// TwinCAT 3 PLC project Untitled1
// ProgramVersion: 3.1.4024.0
// libraries:
//   Tc2_Standard, * (Beckhoff Automation GmbH)
//   Tc2_System, * (Beckhoff Automation GmbH)
//   Tc3_Module, * (Beckhoff Automation GmbH)
// project tree:
//   / GlobalTextList.TcGTLO, PlcTask.TcTTO, Visualization Manager.TcVMO (not stored), Visualization.TcVIS
//   GVLs/ GVL.TcGVL
//   POUs/ Brightspace.TcPOU, MotivationAnalysis.TcPOU, Student.TcPOU, Calender.TcPOU
// real-time tasks:
//   TASK PlcTask: cycle T#10ms, priority 20, ADS port 350
//   TASK brightspace: cycle T#10ms, priority 1, ADS port 351
//   TASK Calender: cycle T#10ms, priority 2, ADS port 352

CONFIGURATION Untitled1
    RESOURCE PLC ON TwinCAT3
        TASK PlcTask(INTERVAL := T#10ms, PRIORITY := 20);
        PROGRAM Student WITH PlcTask : Student;
        PROGRAM Brightspace WITH PlcTask : Brightspace;
        PROGRAM Calender WITH PlcTask : Calender;
    END_RESOURCE
END_CONFIGURATION

// ---- GVLs/GVL.TcGVL
{attribute 'qualified_only'}
VAR_GLOBAL
	
	StartPls : BOOL;		//signal student to start doing something
	Day : INT:= 0;			//keeps track of what day it is
	Finished: BOOL := 0;	//student can signal he has finished an assingment
	MainDueIn: INT := 0;	//shows how far you are from the deadline
	Cycle: BOOL;			//shows daycycle
END_VAR

// ---- POUs/Student.TcPOU
PROGRAM Student		//program pretending to be a student
VAR
	MaxMotivation1: INT := 75; 	//maximum amount of motivation the student can have on a given day
	Phone: SR;					//phone saves the signal from brightspace as a notification
	StudentNotification: BOOL;	
	DontWantTo: BOOL;			//shows the student is not going to do the work
	MotTrig: R_TRIG;			
	MotTrigHigh: BOOL;
	Motivation: INT;
	Timer: TON;
	
	MotivationTracker: ARRAY[1..25] OF INT;	//tracks motivation for visualisation
	ArrayCount: INT := 1;					//position in bar graph
END_VAR

//set notification
Phone(SET1:=GVL.StartPls , RESET:=GVL.Finished OR DontWantTo , Q1=>StudentNotification );

//daily motivation calculated each morning :)
MotTrig(CLK:=StudentNotification , Q=>MotTrigHigh );
IF MotTrigHigh = TRUE THEN
	Motivation := MotivationAnalysis(MaxMotivation2:=MaxMotivation1 );
	
	//visualisation fun
	MotivationTracker[ArrayCount] := Motivation;
	ArrayCount := ArrayCount + 1;
	IF ArrayCount > 25 THEN
		ArrayCount := 1;
	END_IF
END_IF

//when the student has a notification pending they will decide what to do with it depending on the amount of motivation they have minus the amount of time they have left to finish it
IF StudentNotification = TRUE THEN
	IF (GVL.MainDueIn*-1) + Motivation > 69 THEN
		GVL.Finished := TRUE;
	ELSIF (GVL.MainDueIn*-1) + Motivation < 69 THEN
		DontWantTo := TRUE;
		Timer(IN := TRUE, PT := T#50MS);
	END_IF
END_IF

//turn DontWantTo off for as long as needed
IF Timer.Q THEN
    DontWantTo := FALSE;
    Timer(IN := FALSE);
END_IF

END_PROGRAM

// ---- POUs/MotivationAnalysis.TcPOU
FUNCTION MotivationAnalysis : INT	//function which gives a random number between 0 and the max value
VAR_INPUT
	MaxMotivation2: INT;
END_VAR
VAR
	Roll4Motivation: DRAND;
	RandomReal: LREAL;
END_VAR

//DRAND function with daynumber as seed
Roll4Motivation(Seed:=GVL.Day , Num=>RandomReal );

//changes the range from 0-1 to 1-whatever you put as maximum
MotivationAnalysis := 1 + LREAL_TO_INT (RandomReal * MaxMotivation2);

END_FUNCTION

// ---- POUs/Brightspace.TcPOU
PROGRAM Brightspace		//program pretending to be brightspace
VAR
	TaskMaster: ARRAY[1..3] OF INT := [
        0, 0, 1    // 30 day task
    ];
	TasksGiven: INT;	
	Late: BOOL;
END_VAR

//how many days till certain assignment needs to be done
GVL.MainDueIn := TaskMaster[2] - GVL.Day;

//make task
IF TaskMaster[1] = 0 OR GVL.MainDueIn < 1 AND TaskMaster[3] = 1 THEN
	GVL.Finished := FALSE;
	TaskMaster[1] := TasksGiven + 1;
	TaskMaster[2] := GVL.Day + 30;
	TaskMaster[3] := 0;
	TasksGiven := TasksGiven +1;
	GVL.StartPls := TRUE;
END_IF

//arrays and global variables dont mix
IF GVL.Finished = TRUE THEN				//yes im using this if statement as an SR flipflop
	TaskMaster[3] := 1;
END_IF
 
//send signal once to remind the student to pls start doing something
IF GVL.MainDueIn = 30 AND TaskMaster[3] = 0 OR GVL.MainDueIn = 20 AND TaskMaster[3] = 0 OR GVL.MainDueIn = 10 AND TaskMaster[3] = 0 OR GVL.MainDueIn <= 1 AND TaskMaster[3] = 0 THEN 
	GVL.StartPls := TRUE;
	IF GVL.MainDueIn <0 AND TaskMaster[3] = 0 THEN
		GVL.StartPls := GVL.Cycle;
	END_IF
ELSE
	GVL.StartPls := FALSE;		
END_IF 

IF GVL.MainDueIn <0 THEN
	Late := TRUE;
ELSE 
	Late := FALSE;
END_IF

END_PROGRAM

// ---- POUs/Calender.TcPOU
PROGRAM Calender //adjustable on/off timer program
VAR
	DayNight: SR;
	calenderTimer: TON;
	AnotherOne: TON;
	Cycle: BOOL;
	Start: BOOL;
	On: BOOL;			//turn time on/off
	Morning: BOOL;
	HalfADay: TIME := T#1000ms;
END_VAR

calenderTimer(IN:=Start , PT:= HalfADay, Q=> Cycle , ET=> );

IF Cycle = TRUE THEN
	GVL.Day := GVL.Day + 1;
	GVL.Cycle := TRUE;
	Start := FALSE;
ELSE
	GVL.Cycle := FALSE;
END_IF

AnotherOne(IN:=on AND NOT Start , PT:=HalfADay , Q=>Morning , ET=> );

DayNight(SET1:=Morning , RESET:=Cycle , Q1=>Start );

END_PROGRAM

// ---- GlobalTextList.TcGTLO
TEXTLIST GlobalTextList
  496 = ''
  624 = '%brightspace.TasksFinished%'
  487 = '%GVL.TasksFinished%'
  525 = '%TasksCompleted%'
  947 = 'adg'
  597 = 'calender on/off'
  634 = 'Days to finish assignment'
  68 = 'daytime'
  555 = 'Late'
  284 = 'Max. motivation \ncontrol'
  600 = 'Max. motivation control'
  566 = 'Maximum motivation control'
  140 = 'Motivation'
  505 = 'Motivation amount'
  492 = 'Motivation of the last \n25 days where you needed it'
  342 = 'Motivation of the last \n25 days you needed it'
  826 = 'Motivation of the last 25 days you needed it'
  377 = 'Motivation/day'
  563 = 'ms'
  711 = 'Notification'
  557 = 'Speed of time \n0.25s-3s'
  903 = 'Speed of time 0.25s-3s'
  543 = 'start/stop \ntime itself'
  680 = 'start/stop time itself'
  909 = 'task finished'
  857 = 'Time manipulation\n0.25s-3s'
  279 = "[Moti's]"
  845 = "[Moti's] AKA How much motivation you have"
  357 = "[Moti's] AKA motivation amount"
  359 = '[ms]'
  814 = '{brightspace.TasksCompleted}'
  638 = '{brightspace.TasksFinished}'
  759 = '{GVL.Day}'
END_TEXTLIST

// ---- Visualization.TcVIS
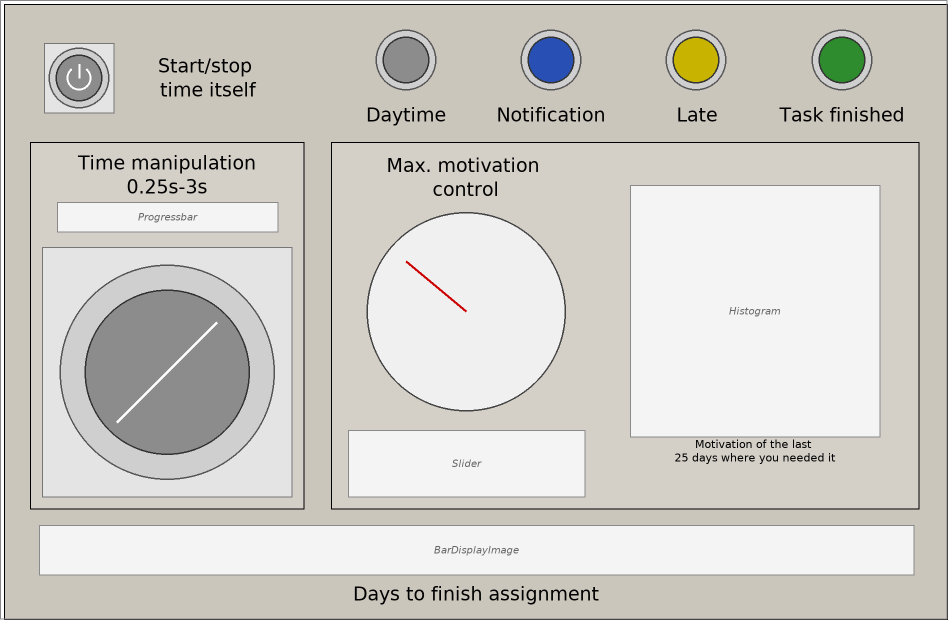
VISUALIZATION Visualization  // 948x620
    Rectangle (4,4 944x616)
    RoundedRectangle (331,142 588x367)
    RoundedRectangle (30,142 274x367)
    Label (133,51 150x54), "Start/stop time itself"
    PowerSwitch (44,43 70x70), variable: Calender.On, behaviour: TOGGLE, style: Switch-PowerSwitch-Gray
    Progressbar (57,202 221x30), variable: Calender.HalfADay
    Label (70,153 194x44), "Time manipulation 0.25s-3s"
    Potentiometer360 (42,247 250x250), variable: Calender.HalfADay, style: Potentiometer-Potentiometer360-Gray, scale format: %.1f, scale 250..2250
        p518627256: [ms]
    Histogram (630,185 250x252), scale format: %.1f, scale 0..100
        p1518820177: Student.MotivationTracker
        p102497268: Student.MotivationTracker
        p788070771: ARRAY [1..25] OF INT
    Label (674,436 162x30), "Motivation of the last 25 days where you needed it"
    Meter360 (363,212 206x199), value: Student.Motivation, style: Meter-Meter360-Gray, scale format: %.1f, scale 0..100
        p518627256: Motivation amount
    Slider (348,430 237x67), variable: Student.MaxMotivation1, scale 0..100
    Label (336,152 260x51), "Max. motivation control"
    Label (331,100 150x30), "Daytime"
    Label (767,100 150x30), "Task finished"
    Label (622,100 150x30), "Late"
    Label (476,100 150x30), "Notification"
    Lamp1 (371,25 70x70), variable: Calender.calenderTimer.IN, style: Lamp-Lamp1-Gray
    Lamp1 (807,25 70x70), variable: GVL.Finished, style: Lamp-Lamp1-Green
    Lamp1 (661,25 70x70), variable: brightspace.Late, style: Lamp-Lamp1-Yellow
    Lamp1 (516,25 70x70), variable: Student.StudentNotification, style: Lamp-Lamp1-Blue
    BarDisplayImage (39,525 875x50), value: GVL.MainDueIn, style: BarDisplayImage-Gray, scale format: %.1f, scale -30..30
    Label (328,579 296x30), "Days to finish assignment"
END_VISUALIZATION
